PROGRAM MAIN
VAR
    originalRectangle: Rectangle;
    clonedRectangle: ITF_Shape;
	
    originalCircle: Circle;
    clonedCircle: ITF_Shape;
	
	bRequest : BOOL;
	counter: INT;

END_VAR

// https://refactoring.guru/design-patterns/prototype

// Recuerda que el patrón Prototipo permite crear nuevos objetos clonando un objeto existente, evitando así la necesidad de crear nuevas instancias desde cero.

// porque salen varios mensajes:
// https://github.com/tcunit/TcUnit/issues/92
// solución temporal : Unload project...

IF bRequest THEN
	
	originalRectangle.width := 10;
	originalRectangle.height := 5;
	originalRectangle.Draw();
	clonedRectangle := originalRectangle.clone();
	clonedRectangle.Draw();
	
	originalCircle.radius := 7;
	originalCircle.Draw();
	clonedCircle := originalCircle.clone();
	clonedCircle.Draw();
		
	bRequest := FALSE;
//	counter := counter + 1;
//	ADSLOGSTR(msgCtrlMask :=ADSLOG_MSGTYPE_HINT, msgFmtStr :='test: %s', strArg := TO_STRING(counter));
END_IF

END_PROGRAM

(* stored: Version 1.1.0.1, ProductVersion 3.1.4024.12
   POU MAIN: Id {6e781358-1f8a-4796-9164-36ac68c8106e}, SpecialFunc None *)
